Yaskawa INFORM job: SKRZYNIA_4040_-90_STOPNI_10BR.JBI

/JOB
//NAME SKRZYNIA_4040_-90_STOPNI_10BR
///FOLDERNAME 02-SKRZYNIE_JOBS
//POS
///NPOS 404,404,0,30,0,0
///TOOL 0
///POSTYPE PULSE
///PULSE
C00000=0,-52280,40443,0,6876,0
C00001=-82314,-24956,17040,-59626,-27382,-6248
C00002=-93910,-8625,17040,-59626,-43355,-6248
C00003=-98846,-1061,-42166,-80308,-57081,16120
C00004=-100452,6057,-48127,-85711,-56704,21322
C00005=-96957,25597,-37888,-85158,-62082,25522
C00006=-95580,33075,-33256,-84644,-64024,26851
C00007=-94380,33739,-32188,-85134,-63496,26721
C00008=-95580,33075,-33256,-84644,-64024,26851
C00009=-94940,31262,-36138,-85248,-63712,27160
C00010=-95580,33075,-33256,-84644,-64024,26851
C00011=-95263,33142,-33256,-84677,-63995,26850
C00012=-95263,33142,-33256,-84677,-63995,26850
C00013=-94261,33702,-32359,-85087,-63552,26740
C00014=-95263,33142,-33256,-84677,-63995,26850
C00015=-94777,31773,-35433,-85135,-63758,27084
C00016=-95263,33142,-33256,-84677,-63995,26850
C00017=-95260,33144,-33256,-84678,-63995,26850
C00018=-95260,33144,-33256,-84678,-63995,26850
C00019=-94282,33689,-32380,-85076,-63563,26742
C00020=-95260,33144,-33256,-84678,-63995,26850
C00021=-94827,31920,-35204,-85086,-63784,27059
C00022=-95260,33144,-33256,-84678,-63995,26850
C00023=-95258,33145,-33257,-84676,-63996,26846
C00024=-95258,33145,-33257,-84676,-63996,26846
C00025=-94286,33686,-32387,-85074,-63568,26738
C00026=-95258,33145,-33257,-84676,-63996,26846
C00027=-94874,32057,-34990,-85039,-63809,27032
C00028=-95258,33145,-33257,-84676,-63996,26846
C00029=-95377,22848,-19980,-77610,-66139,18413
C00030=-95383,22536,-19091,-77284,-66299,17999
C00031=-94454,23123,-18267,-77513,-65785,17889
C00032=-95383,22536,-19091,-77284,-66299,17999
C00033=-94991,21279,-20843,-77511,-66022,18108
C00034=-95383,22536,-19091,-77284,-66299,17999
C00035=-95258,25631,32269,-66559,-75499,2416
C00036=-95258,25631,32269,-66559,-75499,2416
C00037=-94333,26371,33350,-66433,-74983,2224
C00038=-95258,25631,32269,-66559,-75499,2416
C00039=-94886,24142,30119,-66602,-75133,2534
C00040=-95258,25631,32269,-66559,-75499,2416
C00041=-99189,25294,31874,-88720,-76886,6359
C00042=-99241,29593,38161,-92696,-78880,6430
C00043=-98514,30143,38992,-92642,-78372,6377
C00044=-99241,29593,38161,-92696,-78880,6430
C00045=-98973,29806,38536,-92693,-79698,6341
C00046=-99241,29593,38161,-92696,-78880,6430
C00047=-97871,32974,47728,-100928,-77160,11375
C00048=-97482,34142,50625,-102456,-76680,12291
C00049=-96768,34808,51684,-102358,-76154,12246
C00050=-97504,36083,53738,-102448,-77517,11844
C00051=-97263,35860,53475,-102452,-77986,11780
C00052=-97504,36083,53738,-102448,-77517,11844
C00053=-100410,-1172,-854,-105537,-63273,18802
C00054=-79271,-37169,-30482,-103288,-47510,17696
C00055=-79271,-9415,41877,-76443,-46100,-604
C00056=-100699,17246,57649,-91568,-58011,5122
C00057=-100093,19087,27862,-95634,-72730,8691
C00058=-99472,28508,32136,-95947,-79676,10682
C00059=-98577,29153,33099,-95929,-79046,10644
C00060=-99472,28508,32136,-95947,-79676,10682
C00061=-99113,26771,29576,-96019,-79505,10911
C00062=-99472,28508,32136,-95947,-79676,10682
C00063=-99199,18818,35660,-68259,-73735,6208
C00064=-95720,15423,18785,-70454,-68603,10022
C00065=-95720,15423,18785,-70454,-68603,10022
C00066=-97322,30100,38585,-71742,-79662,10416
C00067=-96349,30901,39804,-71630,-79090,10224
C00068=-97322,30100,38585,-71742,-79662,10416
C00069=-97054,28837,36680,-71776,-79387,10556
C00070=-97322,30100,38585,-71742,-79662,10416
C00071=-97373,30352,38967,-71736,-79717,10385
C00072=-97373,30352,38967,-71736,-79717,10385
C00073=-96432,31128,40151,-71627,-79165,10198
C00074=-97373,30352,38967,-71736,-79717,10385
C00075=-97071,28917,36802,-71776,-79407,10544
C00076=-97373,30352,38967,-71736,-79717,10385
C00077=-97356,30262,38827,-71739,-79698,10398
C00078=-97356,30262,38827,-71739,-79698,10398
C00079=-96507,30957,39891,-71642,-79201,10230
C00080=-97356,30262,38827,-71739,-79698,10398
C00081=-97092,29010,36937,-71773,-79425,10538
C00082=-97356,30262,38827,-71739,-79698,10398
C00083=-99745,23507,8579,-87147,-79275,20063
C00084=-99745,23568,9251,-87081,-79277,19867
C00085=-98882,24102,10002,-87178,-78701,19809
C00086=-99745,23568,9251,-87081,-79277,19867
C00087=-99406,22118,7226,-87176,-79050,20009
C00088=-99745,23568,9251,-87081,-79277,19867
C00089=-99071,22682,8038,-99994,-80807,17980
C00090=-99209,25375,15159,-99348,-81562,16520
C00091=-98424,25891,15901,-99427,-81018,16519
C00092=-99209,25375,15159,-99348,-81562,16520
C00093=-98879,23940,13118,-99425,-81414,16690
C00094=-99209,25375,15159,-99348,-81562,16520
C00095=-97630,34865,50283,-105962,-77348,9129
C00096=-97167,37263,56205,-105494,-76312,8157
C00097=-96392,38071,57532,-105366,-75722,8098
C00098=-97167,37263,56205,-105494,-76312,8157
C00099=-96830,35301,53019,-105613,-76328,8514
C00100=-97167,37263,56205,-105494,-76312,8157
C00101=-98819,19954,1043,-111479,-83154,14713
C00102=-100194,5325,-45038,-118611,-84970,27548
C00103=-77958,-36127,-88985,-138175,-66584,26591
C00104=-62749,-65297,-81682,-146767,-31843,20298
C00105=-53629,-59560,-53714,-89083,-24254,-4356
C00106=-73187,-23116,26488,-26118,-57509,-28469
C00107=-96139,-22548,-25766,-67560,-51232,-5154
C00108=-98398,-8109,-25057,-81551,-55130,4513
C00109=-99451,17861,2757,-80571,-73406,6045
C00110=-99056,24650,11359,-80216,-77425,5946
C00111=-98115,25261,12228,-80295,-76818,5843
C00112=-99056,24650,11359,-80216,-77425,5946
C00113=-98800,23560,9817,-80291,-77224,6050
C00114=-99056,24650,11359,-80216,-77425,5946
C00115=-99819,33446,48735,-87787,-79679,-1235
C00116=-99819,33446,48735,-87787,-79679,-1235
C00117=-98945,34179,49898,-87659,-79086,-1350
C00118=-99819,33446,48735,-87787,-79679,-1235
C00119=-99591,32133,46677,-87830,-79529,-1033
C00120=-99819,33446,48735,-87787,-79679,-1235
C00121=-98841,-14263,-23955,-101504,-55644,8170
C00122=-96175,-21848,-39130,-108881,-63715,10829
C00123=-56537,-51855,-41447,-79827,-26849,-3300
///LIMIT ON
C00124=-37962,-64638,6899,-31784,1461,6885
///LIMIT OFF
C00125=0,-43112,23163,32261,-40956,29092
C00126=-38075,-37396,2384,-17964,-21120,46852
C00127=-50509,-19000,10610,-51503,-15997,61182
C00128=-53130,-17211,12007,-56251,-17152,63186
C00129=-51822,-15992,12994,-55136,-16324,62798
C00130=-53635,-15431,13457,-57815,-17251,63894
C00131=-53130,-17211,12007,-56251,-17152,63186
C00132=-50704,-18403,11069,-52157,-16018,61478
C00133=-53231,-16470,14622,-53206,-17893,61673
C00134=-51756,-15101,15744,-51790,-16990,61165
C00135=-53741,-14453,16285,-54808,-17949,62397
C00136=-53231,-17580,11714,-56182,-17246,63139
C00137=-51814,-19410,10295,-53186,-16720,61844
C00138=-53629,-18979,7405,-62018,-16535,65958
C00139=-52238,-17698,8415,-61175,-15613,65699
C00140=-53551,-17401,8655,-62910,-16346,66402
C00141=-52880,-17654,11656,-55678,-17066,62935
C00142=-51005,-17995,11387,-52847,-16122,61778
C00143=-52964,-17611,11689,-55811,-17106,62990
C00144=-51611,-16353,12697,-54642,-16249,62582
C00145=-53495,-15765,13180,-57466,-17201,63739
C00146=-52964,-17611,11689,-55811,-17106,62990
C00147=-51030,-17982,11395,-52891,-16135,61798
C00148=-52975,-17563,11726,-55850,-17109,63009
C00149=-51607,-16289,12749,-54669,-16241,62596
C00150=-53283,-15811,13140,-57177,-17094,63622
C00151=-52975,-17563,11726,-55850,-17109,63009
C00152=-50945,-18019,11363,-52741,-16103,61737
C00153=-52728,-17788,11545,-55393,-17010,62816
C00154=-51045,-16207,12813,-53894,-15944,62287
C00155=-52895,-15647,13274,-56746,-16874,63461
C00156=-52728,-17788,11545,-55393,-17010,62816
C00157=-50945,-18019,11363,-52741,-16103,61737
C00158=-52556,-17520,11756,-55311,-16888,62798
C00159=-51113,-16157,12849,-54025,-15975,62343
C00160=-52730,-15718,13210,-56498,-16792,63358
C00161=-52556,-17520,11756,-55311,-16888,62798
C00162=-50945,-18019,11363,-52741,-16103,61737
C00163=-51893,-17787,11546,-54246,-16568,62356
C00164=-50379,-16341,12703,-52826,-15610,61849
C00165=-52406,-15704,13225,-56071,-16614,63190
C00166=-51893,-17787,11546,-54246,-16568,62356
C00167=-50028,-22953,-3957,-22347,-31919,54220
C00168=-50947,-22502,-3625,-23433,-32061,54736
C00169=-49421,-20951,-2455,-21951,-31329,54057
C00170=-51207,-20433,-2055,-24026,-31698,55041
C00171=-50529,-22709,-3778,-22940,-31995,54502
C00172=-49763,-25421,-36239,-24565,-26935,60445
C00173=-49763,-25421,-36239,-24565,-26935,60445
C00174=-48299,-23485,-34758,-23276,-26122,59713
C00175=-50218,-22723,-34165,-25568,-26529,60993
C00176=-49763,-25421,-36239,-24565,-26935,60445
C00177=-50713,-12366,-58367,-41124,-17813,74400
C00178=-50824,-12254,-58263,-41255,-17847,74484
C00179=-49431,-10052,-56192,-40383,-17131,73813
C00180=-50915,-9358,-55524,-41955,-17664,74847
C00181=-51028,-12852,-58814,-41301,-17980,74542
C00182=-49763,-25421,-36239,-24565,-26935,60445
C00183=-50529,-22709,-3778,-22940,-31995,54502
C00184=-45389,-28224,4312,-35967,-15579,54278
C00185=-40154,-51179,-915,-24203,-8234,36524
C00186=0,-52280,40443,0,6876,0
C00187=-41463,-32191,18163,-91991,-64949,55938
C00188=0,-52277,40442,0,6872,4
C00189=-82314,-24956,17040,-59626,-27382,-6248
C00190=-93910,-8625,17040,-59626,-43355,-6248
C00191=-98846,-1061,-42166,-80308,-57081,16120
C00192=-100452,6057,-48127,-85711,-56704,21322
C00193=-95564,34698,-34234,-85516,-63941,27819
C00194=-94221,34299,-28769,-82558,-65564,25844
C00195=-94107,37241,-30442,-84005,-65307,27544
C00196=-95103,32620,-31323,-83378,-64939,26072
C00197=-95103,32620,-31323,-83378,-64939,26072
C00198=-93990,32828,-31380,-83932,-64473,26160
C00199=-94063,31710,-30585,-83283,-64598,25457
C00200=-96692,32939,-31211,-82617,-65723,26190
C00201=-96111,21840,170,-71736,-70232,11396
C00202=-94229,22391,773,-71789,-70557,11468
C00203=-94283,22521,1025,-71678,-70686,11433
C00204=-95675,19167,-4176,-72970,-68231,11735
C00205=-95681,24338,3488,-71459,-71669,11415
C00206=-94245,22750,1246,-71757,-70674,11453
C00207=-94341,22923,1499,-71729,-70746,11440
C00208=-96213,24222,3324,-71394,-71999,11479
C00209=-95517,23330,2066,-71543,-71508,11507
C00210=-94304,22892,1449,-71738,-70721,11443
C00211=-94158,22889,1452,-71756,-70627,11429
C00212=-96071,24319,3461,-71408,-71916,11455
C00213=-96941,-6406,-33809,-76117,-54125,10511
C00214=-90643,-26862,-25633,-62597,-56791,-1368
C00215=-66103,-61757,7450,-21008,-32955,-5749
C00216=4223,-52290,40457,-5766,6913,3980
C00217=4223,-52290,40457,-5766,6913,3980
C00218=-4825,-36686,24602,37792,-30278,35378
C00219=-46221,-29633,7403,-27051,-24124,46751
C00220=-46221,-29633,7403,-27051,-24124,46751
C00221=-52474,-20611,11454,-41004,-23045,52959
C00222=-60257,-19980,-2088,-84190,-23320,82051
C00223=-63868,-19883,-6318,-95759,-28031,88346
C00224=-51819,-22965,8574,-41365,-22900,53139
C00225=-4825,-36686,24602,37792,-30278,35378
C00226=0,-52280,40443,0,6876,0
C00227=4223,-52290,40457,-5766,6913,3980
C00228=-66103,-61757,7450,-21008,-32955,-5749
C00229=-89093,-33107,-44597,-67545,-52550,2722
C00230=-96941,-6406,-33809,-76117,-54125,10511
C00231=-99429,14378,84,-80785,-71596,8628
C00232=-99699,24313,24829,-82602,-77917,4569
C00233=-98066,26841,20697,-83331,-79245,6860
C00234=-98079,26929,20513,-83349,-79351,6953
C00235=-99638,19663,10292,-84193,-74452,7551
C00236=-98909,20891,5205,-92499,-77779,3679
C00237=-97991,21897,3469,-96150,-79490,1870
C00238=-97094,22407,2872,-101449,-80737,3094
C00239=-98052,22735,7381,-100906,-80646,1724
C00240=-96016,28471,32512,-109475,-77029,-270
C00241=-93697,27731,31018,-109675,-75757,229
C00242=-93697,30712,42128,-108463,-73689,-2160
C00243=-100174,9543,-9646,-113455,-77250,7387
C00244=-100174,1289,-12558,-103866,-68626,6781
C00245=-100177,-4656,-30138,-114506,-71921,12431
C00246=-97546,-19067,-24950,-97028,-60115,5718
C00247=-61441,-38616,11032,-55510,-42874,-3049
C00248=4223,-52290,40457,-5766,6913,3980
C00249=4223,-52290,40457,-5766,6913,3980
C00250=-4825,-36686,24602,37792,-30278,35378
C00251=-46221,-29633,7403,-27051,-24124,46751
C00252=-56796,-22932,368,-68953,-21567,70907
C00253=-61611,-20349,-6598,-95791,-25091,88405
C00254=-62244,-19942,-5791,-95984,-25882,88372
C00255=-57752,-2938,32150,-100764,-20307,82364
C00256=-58257,-11045,22458,-94361,-23082,79795
C00257=-49294,-34086,9663,-30689,-30758,52546
C00258=4223,-52290,40457,-5766,6913,3980
C00259=0,-52280,40443,0,6876,0
C00260=0,-52280,40443,0,6876,0
C00261=-61754,-61602,7279,-16215,-32140,-7126
C00262=-89313,-24027,20291,-53466,-58905,-4975
C00263=-97807,-25409,-21837,-78881,-62828,2121
C00264=-100103,-15040,-13507,-79140,-58253,2724
C00265=-99725,9645,23361,-67154,-68568,-2059
C00266=-99271,16305,34765,-72797,-70067,-2351
C00267=-98402,25140,29245,-92090,-76944,4625
C00268=-98402,28265,40696,-90956,-76523,2010
C00269=-98754,23130,28932,-98122,-73671,5428
C00270=-98112,-9349,-13739,-99107,-55531,8873
C00271=-87692,-34175,-39658,-96739,-43399,8225
C00272=-75165,-16680,32803,-38944,-52307,-27215
C00273=-75165,-16680,32803,-38944,-52307,-27215
C00274=-96391,11374,61850,-52875,-60261,-22353
C00275=-96391,-17993,-25254,-79577,-45337,-1997
C00276=-84714,-13514,-21320,-79690,-37366,-2300
C00277=-92093,-5454,-13554,-80916,-52292,-613
C00278=-99761,24721,23429,-79408,-77929,-316
C00279=-99564,24916,23930,-79374,-77823,-417
C00280=-100005,27069,23687,-81767,-79755,895
C00281=-97295,30454,38512,-73622,-79542,-3831
C00282=-98471,27958,25022,-81751,-79627,782
C00283=-99805,23386,18402,-82055,-77455,1200
C00284=-100093,24719,20298,-81968,-77939,1081
C00285=-98451,26404,20171,-83400,-79044,-389
C00286=-98528,26732,19657,-84000,-79459,-654
C00287=-100109,23919,19160,-82044,-77303,1139
C00288=-98037,-4340,-16930,-86109,-58746,2389
C00289=-93345,-31758,-40240,-83703,-37467,-946
C00290=-81087,-35886,-14825,-53529,-36311,-18004
C00291=-47029,-49867,-20464,-11808,-29290,-36568
///LIMIT ON
C00292=-41431,-67449,10869,-1325,127,-6150
///LIMIT OFF
C00293=6328,-52297,40483,-8599,6957,5944
C00294=6328,-52297,40483,-8599,6957,5944
C00295=-10231,-60460,6271,71658,-11927,-13637
C00296=-49129,-39322,3023,-34904,-18609,43900
C00297=-57258,-19535,13114,-46502,-25798,55150
C00298=-58736,-19151,1344,-78268,-22199,76919
C00299=-56868,-17231,8572,-62431,-21728,66645
C00300=-56011,-29317,6725,-41009,-27363,52457
C00301=-10137,-60963,4526,62308,-14518,-6745
C00302=0,-52280,40443,0,6876,0
C00303=0,-52280,40443,0,6876,0
C00304=-41653,-63035,2931,-3578,-7576,-14589
C00305=-45770,-50109,-20524,-10089,-29273,-37310
C00306=-80544,-36303,-15042,-52975,-36116,-18265
C00307=-93028,-32302,-40599,-83495,-37263,-1079
C00308=-98446,-3141,-15678,-86094,-59021,2414
C00309=-99951,24070,19376,-82000,-77829,1145
C00310=-98655,27908,24922,-81730,-79774,792
C00311=-98593,28720,26118,-81685,-80145,709
C00312=-99951,24070,19376,-82000,-77829,1145
C00313=-99951,24070,19376,-82000,-77829,1145
C00314=-98577,27118,23759,-81796,-79157,859
C00315=-98518,28577,26461,-81649,-79882,537
C00316=-99951,24070,19376,-82000,-77829,1145
C00317=-100023,27130,33022,-92975,-78123,-161
C00318=-98580,26185,31637,-93003,-77167,-1
C00319=-98580,30404,46303,-91600,-76541,-3267
C00320=-100724,18056,24349,-92081,-73134,-455
C00321=-98404,-4962,-6255,-93190,-58383,1895
C00322=-99487,-12045,-28221,-93829,-57357,5545
C00323=-95086,-30272,-46998,-91958,-53375,4609
C00324=-81694,-37220,-20464,-64791,-45723,-12569
C00325=-45770,-50109,-20524,-10089,-29273,-37310
///LIMIT ON
C00326=-40984,-65135,6743,-2520,-4051,-10897
///LIMIT OFF
C00327=0,-52280,40443,0,6876,0
C00328=0,-52280,40443,0,6876,0
///LIMIT ON
C00329=-50974,-46557,23391,-77768,-13896,42026
///LIMIT OFF
C00330=-53474,-39983,4253,-39182,-18848,44272
C00331=-56619,-19856,12878,-45665,-25558,54806
C00332=-53298,-26712,-11188,-26889,-32979,52528
C00333=-57200,-20845,-7559,-37425,-33513,53351
C00334=-58648,-23818,-25853,-45100,-31207,62168
C00335=-58477,-22145,-38977,-48305,-29254,64725
C00336=-51868,-27423,-11673,-25269,-32728,51737
C00337=-49121,-45409,-2608,-26656,-19965,38583
C00338=-21301,-61008,4568,43957,-10534,-712
C00339=0,-52280,40443,0,6876,0
C00340=0,-52280,40443,0,6876,0
///LIMIT ON
C00341=-40221,-67507,11044,-1325,-65,-6716
///LIMIT OFF
C00342=-45770,-50109,-20525,-10088,-29274,-37311
C00343=-80544,-36303,-15042,-52975,-36116,-18265
C00344=-93028,-32301,-40599,-83495,-37262,-1079
C00345=-97841,-4898,-17503,-86112,-58614,2374
C00346=-97574,22325,42435,-102650,-66613,-1893
C00347=-95754,35899,57018,-103970,-74003,-2798
C00348=-95754,43745,77672,-101743,-71699,-6650
C00349=-99714,17597,9613,-108150,-76803,6279
C00350=-93796,-17226,-33718,-118170,-55432,13587
C00351=-66816,-54797,-57006,-119089,-33370,13303
C00352=-66816,-52758,-50486,-115256,-31854,11154
C00353=-98141,-7636,2315,-105626,-50514,3722
C00354=-99521,20918,46679,-89083,-66665,-5358
C00355=-98691,34973,58126,-90608,-76643,-4580
C00356=-98691,42061,76615,-89053,-76304,-8086
C00357=-98720,15018,65588,-59406,-66947,-17238
C00358=-93628,-24224,-10838,-81898,-52333,-4131
C00359=-86170,-37737,-28198,-69261,-47898,-9342
C00360=-45770,-50109,-20525,-10088,-29274,-37311
///LIMIT ON
C00361=-40221,-67507,11044,-1325,-65,-6716
///LIMIT OFF
C00362=0,-52280,40443,0,6876,0
C00363=0,-52280,40443,0,6876,0
///LIMIT ON
C00364=-50971,-46557,23390,-77766,-13895,42026
///LIMIT OFF
C00365=-53475,-39984,4253,-39182,-18848,44273
C00366=-56619,-19856,12878,-45665,-25558,54806
C00367=-57643,-27958,-8553,-51854,-24771,59787
C00368=-66195,-24410,-19095,-90567,-31132,85904
C00369=-63290,-24193,-14362,-80030,-27547,78073
C00370=-39040,-40975,-15408,-18643,-21575,44866
C00371=-11647,-69843,-10959,56399,-11165,-4616
C00372=-15394,-57237,30542,-10392,5525,8219
C00373=0,-52280,40443,0,6876,0
C00374=0,-52280,40443,0,6876,0
///LIMIT ON
C00375=-40221,-67507,11044,-1325,-65,-6716
///LIMIT OFF
C00376=-45770,-50109,-20525,-10088,-29274,-37311
C00377=-95022,-19559,-3970,-66108,-42168,-11789
C00378=-84972,-7110,7117,-67721,-41324,-10731
C00379=-83869,-8155,6098,-67213,-40658,-10968
C00380=-99927,23961,20220,-85683,-78298,772
C00381=-98562,26853,28284,-85090,-78334,-823
C00382=-98562,24944,18750,-86001,-78172,1594
C00383=-99530,24174,17652,-85964,-78826,1685
C00384=-98491,25445,31196,-89357,-76395,-673
C00385=-98197,26014,32882,-93044,-76072,-339
C00386=-99839,23064,19027,-85806,-76881,822
C00387=-86774,-13232,-16630,-85484,-41019,-1154
C00388=-97999,-21060,-29835,-88214,-48653,956
C00389=-98846,-3268,25064,-74217,-51189,-12584
C00390=-70313,-35289,-4922,-51188,-38634,-20596
C00391=-81694,-37221,-20464,-64791,-45723,-12569
C00392=-45770,-50109,-20525,-10088,-29274,-37311
C00393=-41628,-63095,3038,-3547,-7472,-14475
C00394=4223,-52290,40457,-5766,6913,3980
///LIMIT ON
C00395=-50971,-46557,23390,-77766,-13895,42026
///LIMIT OFF
C00396=-53475,-39984,4253,-39182,-18848,44273
C00397=-56619,-19856,12878,-45665,-25558,54806
C00398=-53891,-17708,14512,-43170,-23995,53902
C00399=-60674,-17500,6427,-71116,-24772,71097
C00400=-63181,-17997,2063,-82122,-26831,78394
C00401=-39402,-27697,7664,-17904,-21663,43170
C00402=-11647,-69843,-10959,56399,-11165,-4616
C00403=0,-52280,40443,0,6876,0
BC00000=372198
BC00001=352964
BC00002=352964
BC00003=406723
BC00004=352964
BC00005=352964
BC00006=352964
BC00007=352964
BC00008=352964
BC00009=352964
BC00010=352964
BC00011=399066
BC00012=399066
BC00013=399066
BC00014=399066
BC00015=399066
BC00016=399066
BC00017=445276
BC00018=445276
BC00019=445276
BC00020=445276
BC00021=445276
BC00022=445276
BC00023=491380
BC00024=491380
BC00025=491380
BC00026=491380
BC00027=491380
BC00028=491380
BC00029=481377
BC00030=480887
BC00031=480887
BC00032=480887
BC00033=480888
BC00034=480887
BC00035=467227
BC00036=467227
BC00037=467227
BC00038=467227
BC00039=467227
BC00040=467227
BC00041=464142
BC00042=463563
BC00043=463563
BC00044=463563
BC00045=463563
BC00046=463563
BC00047=467130
BC00048=467852
BC00049=467852
BC00050=467852
BC00051=467852
BC00052=467852
BC00053=431056
BC00054=431056
BC00055=478309
BC00056=512702
BC00057=523223
BC00058=534753
BC00059=534753
BC00060=534753
BC00061=534753
BC00062=534753
BC00063=621951
BC00064=621951
BC00065=621951
BC00066=621951
BC00067=621951
BC00068=621951
BC00069=621951
BC00070=621951
BC00071=645037
BC00072=645037
BC00073=645037
BC00074=645037
BC00075=645037
BC00076=645037
BC00077=691109
BC00078=691109
BC00079=691109
BC00080=691109
BC00081=691109
BC00082=691109
BC00083=714198
BC00084=714198
BC00085=714197
BC00086=714198
BC00087=714198
BC00088=714198
BC00089=721422
BC00090=721422
BC00091=721422
BC00092=721422
BC00093=721422
BC00094=721422
BC00095=705839
BC00096=705839
BC00097=705839
BC00098=705839
BC00099=705839
BC00100=705839
BC00101=706227
BC00102=715152
BC00103=741215
BC00104=815410
BC00105=809921
BC00106=799182
BC00107=831839
BC00108=838454
BC00109=838479
BC00110=838485
BC00111=838485
BC00112=838485
BC00113=838485
BC00114=838485
BC00115=819448
BC00116=834809
BC00117=834809
BC00118=834809
BC00119=834809
BC00120=834809
BC00121=835662
BC00122=825379
BC00123=817159
BC00124=681039
BC00125=719629
BC00126=804722
BC00127=797458
BC00128=797458
BC00129=797458
BC00130=797458
BC00131=797458
BC00132=736016
BC00133=736016
BC00134=736016
BC00135=736016
BC00136=736016
BC00137=674586
BC00138=674586
BC00139=674586
BC00140=674586
BC00141=674586
BC00142=613184
BC00143=613184
BC00144=613184
BC00145=613184
BC00146=613184
BC00147=551699
BC00148=551699
BC00149=551699
BC00150=551699
BC00151=551699
BC00152=490298
BC00153=490298
BC00154=490298
BC00155=490298
BC00156=490298
BC00157=428826
BC00158=428826
BC00159=428826
BC00160=428826
BC00161=428826
BC00162=367374
BC00163=367374
BC00164=367374
BC00165=367374
BC00166=367374
BC00167=367378
BC00168=367378
BC00169=367378
BC00170=367378
BC00171=367378
BC00172=367378
BC00173=367378
BC00174=367378
BC00175=367378
BC00176=367378
BC00177=367378
BC00178=367378
BC00179=367378
BC00180=367378
BC00181=367378
BC00182=367378
BC00183=367378
BC00184=367374
BC00185=441050
BC00186=441050
BC00187=791478
BC00188=382983
BC00189=352964
BC00190=352964
BC00191=408260
BC00192=352964
BC00193=352964
BC00194=353544
BC00195=352960
BC00196=353556
BC00197=391964
BC00198=400011
BC00199=389600
BC00200=400107
BC00201=381081
BC00202=388397
BC00203=381081
BC00204=388818
BC00205=427172
BC00206=434877
BC00207=427169
BC00208=427169
BC00209=457913
BC00210=457913
BC00211=450237
BC00212=450041
BC00213=414344
BC00214=450041
BC00215=427058
BC00216=450041
BC00217=400994
BC00218=490644
BC00219=563016
BC00220=563016
BC00221=563016
BC00222=563016
BC00223=624162
BC00224=624476
BC00225=490644
BC00226=400994
BC00227=450041
BC00228=450041
BC00229=413692
BC00230=498778
BC00231=464973
BC00232=451598
BC00233=459057
BC00234=451696
BC00235=459288
BC00236=477534
BC00237=485795
BC00238=485795
BC00239=485795
BC00240=461742
BC00241=461742
BC00242=461742
BC00243=461742
BC00244=464778
BC00245=461044
BC00246=455085
BC00247=441558
BC00248=492251
BC00249=528027
BC00250=720637
BC00251=795617
BC00252=805108
BC00253=808590
BC00254=827541
BC00255=790719
BC00256=786930
BC00257=760893
BC00258=450041
BC00259=450041
BC00260=450041
BC00261=450041
BC00262=509147
BC00263=545841
BC00264=541316
BC00265=532881
BC00266=530910
BC00267=529272
BC00268=529272
BC00269=529176
BC00270=533263
BC00271=538121
BC00272=540993
BC00273=589567
BC00274=589567
BC00275=648537
BC00276=648537
BC00277=648537
BC00278=648537
BC00279=617841
BC00280=617841
BC00281=611605
BC00282=617971
BC00283=617841
BC00284=634993
BC00285=633229
BC00286=640873
BC00287=640937
BC00288=640937
BC00289=640937
BC00290=640937
BC00291=640937
BC00292=640937
BC00293=640937
BC00294=528027
BC00295=469376
BC00296=406602
BC00297=315730
BC00298=315726
BC00299=376881
BC00300=377231
BC00301=431999
BC00302=431999
BC00303=640937
BC00304=640937
BC00305=640937
BC00306=640937
BC00307=640937
BC00308=640937
BC00309=679258
BC00310=679258
BC00311=687013
BC00312=679258
BC00313=702338
BC00314=702338
BC00315=709052
BC00316=702338
BC00317=697065
BC00318=697065
BC00319=697065
BC00320=699422
BC00321=702188
BC00322=721854
BC00323=728490
BC00324=748432
BC00325=703131
BC00326=649416
BC00327=640936
BC00328=580559
BC00329=483911
BC00330=372992
BC00331=315730
BC00332=315730
BC00333=315730
BC00334=315730
BC00335=315730
BC00336=315730
BC00337=379280
BC00338=431999
BC00339=431999
BC00340=640937
BC00341=640937
BC00342=640937
BC00343=640937
BC00344=640937
BC00345=640937
BC00346=690236
BC00347=698481
BC00348=698481
BC00349=700031
BC00350=700031
BC00351=700031
BC00352=758299
BC00353=758299
BC00354=755546
BC00355=768208
BC00356=768208
BC00357=768208
BC00358=750310
BC00359=761341
BC00360=703131
BC00361=640937
BC00362=640937
BC00363=580559
BC00364=483911
BC00365=421515
BC00366=442691
BC00367=465804
BC00368=465286
BC00369=526143
BC00370=526236
BC00371=526236
BC00372=526236
BC00373=526236
BC00374=640937
BC00375=640937
BC00376=823629
BC00377=816144
BC00378=816144
BC00379=816144
BC00380=839508
BC00381=839510
BC00382=839510
BC00383=839510
BC00384=839617
BC00385=839617
BC00386=840477
BC00387=836719
BC00388=828295
BC00389=807430
BC00390=790908
BC00391=748432
BC00392=703131
BC00393=656709
BC00394=640937
BC00395=657676
BC00396=664515
BC00397=684473
BC00398=684473
BC00399=684473
BC00400=746207
BC00401=745829
BC00402=704594
BC00403=650116
///POSTYPE BASE
///RECTAN
///RCONF 1,0,0,0,0,0,0,0,0,0,0,0,0,0,0,0,0,0,0,0,0,0,0,0
P00006=0.000,0.000,0.000,0.0000,0.0000,0.0000
///RCONF 0,0,0,0,0,0,0,0,0,0,0,0,0,0,0,0,0,0,0,0,0,0,0,0
P00058=0.000,0.000,3.000,0.0000,0.0000,0.0000
///RCONF 1,0,0,0,0,0,0,0,0,0,0,0,0,0,0,0,0,0,0,0,0,0,0,0
P00300=-0.036,-1.505,2.318,0.0000,0.0000,0.0000
P00301=0.046,-2.112,7.779,0.0000,0.0000,0.0000
P00302=-0.180,-2.409,6.326,0.0000,0.0000,0.0000
///RCONF 0,0,0,0,0,0,0,0,0,0,0,0,0,0,0,0,0,0,0,0,0,0,0,0
P00303=-0.004,-1.437,-4.584,0.0000,0.0000,0.0000
P00304=0.028,-1.666,-4.234,0.0000,0.0000,0.0000
P00305=-0.003,-1.920,-3.501,0.0000,0.0000,0.0000
P00306=0.015,-2.252,-3.054,0.0000,0.0000,0.0000
P00307=0.019,-2.151,-5.077,0.0000,0.0000,0.0000
P00308=-0.003,-2.092,-4.888,0.0000,0.0000,0.0000
P00309=-0.040,-2.205,-4.992,0.0000,0.0000,0.0000
P00310=-0.006,-2.490,-5.925,0.0000,0.0000,0.0000
P00311=-0.007,-2.079,-5.307,0.0000,0.0000,0.0000
P00312=-0.032,2.202,-7.632,0.0000,0.0000,0.0000
///RCONF 1,0,0,0,0,0,0,0,0,0,0,0,0,0,0,0,0,0,0,0,0,0,0,0
P00313=-0.088,1.055,2.110,0.0000,0.0000,0.0000
P00314=-0.055,1.752,1.634,0.0000,0.0000,0.0000
P00316=0.009,2.112,2.075,0.0000,0.0000,0.0000
P00317=-0.015,2.781,3.126,0.0000,0.0000,0.0000
///RCONF 0,0,0,0,0,0,0,0,0,0,0,0,0,0,0,0,0,0,0,0,0,0,0,0
P00351=13.563,-0.027,-0.653,0.0000,0.0000,0.0000
P00352=13.252,-0.027,-0.827,0.0000,0.0000,0.0000
P00353=10.971,-0.082,0.776,0.0000,0.0000,0.0000
P00354=-0.024,2.508,-1.824,0.0000,0.0000,0.0000
P00355=-0.001,2.528,-1.131,0.0000,0.0000,0.0000
P00356=-0.034,2.921,-0.262,0.0000,0.0000,0.0000
P00357=0.003,3.386,-0.091,0.0000,0.0000,0.0000
P00358=0.014,3.037,-0.020,0.0000,0.0000,0.0000
P00359=-0.005,2.731,0.912,0.0000,0.0000,0.0000
P00360=-0.011,3.412,0.438,0.0000,0.0000,0.0000
P00361=0.018,3.050,1.253,0.0000,0.0000,0.0000
//INST
///DATE 2025/03/25 11:13
///ATTR SC,RW
///GROUP1 RB1,BS1
NOP
CALL JOB:MOVE_INTO_TUNNEL
MOVJ C00000 BC00000 VJ=50.00
MOVJ C00001 BC00001 VJ=40.00
MOVJ C00002 BC00002 VJ=40.00
MOVL C00003 BC00003 V=666.7
COMM MOVJ C00004 BC00004 VJ=30.00
COMM MOVL C00005 BC00005 V=500.0
COMM '------------------------
COMM 'W31.2
COMM '------------------------
COMM MOVL C00006 BC00006 V=166.7 PL=0
COMM REFP 3 C00007 BC00007
COMM CALL JOB:SEARCH-R1
COMM SET P0300 P0006
COMM SFTON P0300
COMM MOVL C00008 BC00008 V=166.7 PL=0
COMM REFP 3 C00009 BC00009
COMM CALL JOB:SEARCH-R1
COMM SET P0300 P0006
COMM SFTON P0300
COMM MOVL C00010 BC00010 V=166.7 PL=0
COMM SFTOF
COMM '------------------------
COMM 'W31.4
COMM '------------------------
COMM MOVL C00011 BC00011 V=500.0
COMM MOVL C00012 BC00012 V=166.7 PL=0
COMM REFP 3 C00013 BC00013
COMM CALL JOB:SEARCH-R1
COMM SET P0301 P0006
COMM SFTON P0301
COMM MOVL C00014 BC00014 V=166.7 PL=0
COMM REFP 3 C00015 BC00015
COMM CALL JOB:SEARCH-R1
COMM SET P0301 P0006
COMM SFTON P0301
COMM MOVL C00016 BC00016 V=166.7 PL=0
COMM SFTOF
'------------------------
'W31.6
'------------------------
MOVL C00017 BC00017 V=500.0
MOVL C00018 BC00018 V=166.7 PL=0
REFP 3 C00019 BC00019
CALL JOB:SEARCH-R1
SET P0302 P0006
SFTON P0302
MOVL C00020 BC00020 V=166.7 PL=0
REFP 3 C00021 BC00021
CALL JOB:SEARCH-R1
SET P0302 P0006
SFTON P0302
MOVL C00022 BC00022 V=166.7 PL=0
SFTOF
'------------------------
'W31.8
'------------------------
MOVL C00023 BC00023 V=500.0
MOVL C00024 BC00024 V=166.7 PL=0
REFP 3 C00025 BC00025
CALL JOB:SEARCH-R1
SET P0303 P0006
SFTON P0303
MOVL C00026 BC00026 V=166.7 PL=0
REFP 3 C00027 BC00027
CALL JOB:SEARCH-R1
SET P0303 P0006
SFTON P0303
MOVL C00028 BC00028 V=166.7 PL=0
SFTOF
'------------------------
'W31.9
'------------------------
MOVL C00029 BC00029 V=500.0
MOVL C00030 BC00030 V=166.7 PL=0
REFP 3 C00031 BC00031
CALL JOB:SEARCH-R1
SET P0304 P0006
SFTON P0304
MOVL C00032 BC00032 V=166.7 PL=0
REFP 3 C00033 BC00033
CALL JOB:SEARCH-R1
SET P0304 P0006
SFTON P0304
MOVL C00034 BC00034 V=166.7 PL=0
SFTOF
'------------------------
'W31.11
'------------------------
MOVL C00035 BC00035 V=500.0
MOVL C00036 BC00036 V=166.7 PL=0
REFP 3 C00037 BC00037
CALL JOB:SEARCH-R1
SET P0305 P0006
SFTON P0305
MOVL C00038 BC00038 V=166.7 PL=0
REFP 3 C00039 BC00039
CALL JOB:SEARCH-R1
SET P0305 P0006
SFTON P0305
MOVL C00040 BC00040 V=166.7 PL=0
SFTOF
'------------------------
'W31.13
'------------------------
MOVL C00041 BC00041 V=500.0
MOVL C00042 BC00042 V=166.7 PL=0
REFP 3 C00043 BC00043
CALL JOB:SEARCH-R1
SET P0306 P0006
SFTON P0306
MOVL C00044 BC00044 V=166.7 PL=0
REFP 3 C00045 BC00045
CALL JOB:SEARCH-R1
SET P0306 P0006
SFTON P0306
MOVL C00046 BC00046 V=166.7 PL=0
SFTOF
'------------------------
'W31.14
'------------------------
MOVL C00047 BC00047 V=333.3
MOVL C00048 BC00048 V=166.7 PL=0
REFP 3 C00049 BC00049
CALL JOB:SEARCH-R1
SET P0307 P0006
SFTON P0307
MOVL C00050 BC00050 V=166.7 PL=0
REFP 3 C00051 BC00051
CALL JOB:SEARCH-R1
SET P0307 P0006
SFTON P0307
MOVL C00052 BC00052 V=166.7 PL=0
SFTOF
MOVL C00053 BC00053 V=500.0
MOVL C00054 BC00054 V=500.0
MOVL C00055 BC00055 V=500.0
MOVL C00056 BC00056 V=500.0
'------------------------
'W31.16
'------------------------
MOVL C00057 BC00057 V=500.0
MOVL C00058 BC00058 V=166.7 PL=0
REFP 3 C00059 BC00059
CALL JOB:SEARCH-R1
SET P0308 P0006
SFTON P0308
MOVL C00060 BC00060 V=166.7 PL=0
REFP 3 C00061 BC00061
CALL JOB:SEARCH-R1
SET P0308 P0006
SFTON P0308
MOVL C00062 BC00062 V=166.7 PL=0
SFTOF
MOVL C00063 BC00063 V=500.0
MOVL C00064 BC00064 V=333.3
'------------------------
'W31.18
'------------------------
MOVL C00065 BC00065 V=166.7
MOVL C00066 BC00066 V=133.3 PL=0
REFP 3 C00067 BC00067
CALL JOB:SEARCH-R1
SET P0309 P0006
SFTON P0309
MOVL C00068 BC00068 V=66.7 PL=0
REFP 3 C00069 BC00069
CALL JOB:SEARCH-R1
SET P0309 P0006
SFTON P0309
MOVL C00070 BC00070 V=66.7 PL=0
SFTOF
'------------------------
'W31.19
'------------------------
MOVL C00071 BC00071 V=500.0
MOVL C00072 BC00072 V=166.7 PL=0
REFP 3 C00073 BC00073
CALL JOB:SEARCH-R1
SET P0310 P0006
SFTON P0310
MOVL C00074 BC00074 V=166.7 PL=0
REFP 3 C00075 BC00075
CALL JOB:SEARCH-R1
SET P0310 P0006
SFTON P0310
MOVL C00076 BC00076 V=166.7 PL=0
SFTOF
'------------------------
'W31.21
'------------------------
MOVL C00077 BC00077 V=500.0
MOVL C00078 BC00078 V=166.7 PL=0
REFP 3 C00079 BC00079
CALL JOB:SEARCH-R1
SET P0311 P0006
SFTON P0311
MOVL C00080 BC00080 V=166.7 PL=0
REFP 3 C00081 BC00081
CALL JOB:SEARCH-R1
SET P0311 P0006
SFTON P0311
MOVL C00082 BC00082 V=166.7 PL=0
SFTOF
'------------------------
'W31.22
'------------------------
MOVL C00083 BC00083 V=500.0
MOVL C00084 BC00084 V=166.7 PL=0
REFP 3 C00085 BC00085
CALL JOB:SEARCH-R1
SET P0312 P0006
SFTON P0312
MOVL C00086 BC00086 V=166.7 PL=0
REFP 3 C00087 BC00087
CALL JOB:SEARCH-R1
SET P0312 P0006
SFTON P0312
MOVL C00088 BC00088 V=166.7 PL=0
SFTOF
'------------------------
'W31.24
'------------------------
MOVL C00089 BC00089 V=500.0
MOVL C00090 BC00090 V=166.7 PL=0
REFP 3 C00091 BC00091
CALL JOB:SEARCH-R1
SET P0313 P0006
SFTON P0313
MOVL C00092 BC00092 V=166.7 PL=0
REFP 3 C00093 BC00093
CALL JOB:SEARCH-R1
SET P0313 P0006
SFTON P0313
MOVL C00094 BC00094 V=166.7 PL=0
SFTOF
'------------------------
'W31.26
'------------------------
MOVL C00095 BC00095 V=500.0
MOVL C00096 BC00096 V=166.7 PL=0
REFP 3 C00097 BC00097
CALL JOB:SEARCH-R1
SET P0314 P0006
SFTON P0314
MOVL C00098 BC00098 V=166.7 PL=0
REFP 3 C00099 BC00099
CALL JOB:SEARCH-R1
SET P0314 P0006
SFTON P0314
MOVL C00100 BC00100 V=166.7 PL=0
SFTOF
'------------------------
MOVL C00101 BC00101 V=333.3
MOVL C00102 BC00102 V=666.7
MOVL C00103 BC00103 V=666.7
MOVL C00104 BC00104 V=666.7
MOVL C00105 BC00105 V=500.0
MOVL C00106 BC00106 V=666.7
MOVL C00107 BC00107 V=666.7
MOVL C00108 BC00108 V=333.3
MOVL C00109 BC00109 V=250.0
'------------------------
'W31.29
'------------------------
MOVL C00110 BC00110 V=166.7 PL=0
REFP 3 C00111 BC00111
CALL JOB:SEARCH-R1
SET P0316 P0006
SFTON P0316
MOVL C00112 BC00112 V=166.7 PL=0
REFP 3 C00113 BC00113
CALL JOB:SEARCH-R1
SET P0316 P0006
SFTON P0316
MOVL C00114 BC00114 V=166.7 PL=0
SFTOF
'------------------------
'W31.31
'------------------------
MOVL C00115 BC00115 V=500.0
MOVL C00116 BC00116 V=166.7 PL=0
REFP 3 C00117 BC00117
CALL JOB:SEARCH-R1
SET P0317 P0006
SFTON P0317
MOVL C00118 BC00118 V=166.7 PL=0
REFP 3 C00119 BC00119
CALL JOB:SEARCH-R1
SET P0317 P0006
SFTON P0317
MOVL C00120 BC00120 V=166.7 PL=0
SFTOF
'------------------------
'W31.32
'------------------------
MOVL C00121 BC00121 V=333.3
MOVL C00122 BC00122 V=333.3
MOVL C00123 BC00123 V=666.7
MOVJ C00124 BC00124 VJ=50.00
MOVJ C00125 BC00125 VJ=50.00
MOVJ C00126 BC00126 VJ=50.00
'W214A P
'------------------------
MOVJ C00127 BC00127 VJ=40.00
MOVL C00128 BC00128 V=166.7 PL=0
REFP 3 C00129 BC00129
CALL JOB:SEARCH-R1
IMOV P0058 V=16.7
SET P0351 P0006
SFTON P0351
REFP 3 C00130 BC00130
CALL JOB:SEARCH-R1
SET P0351 P0006
SFTON P0351
MOVL C00131 BC00131 V=166.7 PL=0
SFTOF
'------------------------
'W219B L
'------------------------
MOVJ C00132 BC00132 VJ=40.00
MOVL C00133 BC00133 V=166.7 PL=0
REFP 3 C00134 BC00134
CALL JOB:SEARCH-R1
IMOV P0058 V=16.7
SET P0352 P0006
SFTON P0352
REFP 3 C00135 BC00135
CALL JOB:SEARCH-R1
SET P0352 P0006
SFTON P0352
MOVL C00136 BC00136 V=166.7 PL=0
SFTOF
'------------------------
'W219B P
'------------------------
MOVJ C00137 BC00137 VJ=40.00
MOVL C00138 BC00138 V=166.7 PL=0
REFP 3 C00139 BC00139
CALL JOB:SEARCH-R1
IMOV P0058 V=16.7
SET P0353 P0006
SFTON P0353
REFP 3 C00140 BC00140
CALL JOB:SEARCH-R1
SET P0353 P0006
SFTON P0353
MOVL C00141 BC00141 V=166.7 PL=0
SFTOF
'------------------------
'W213B L
'------------------------
MOVJ C00142 BC00142 VJ=40.00
MOVL C00143 BC00143 V=166.7 PL=0
REFP 3 C00144 BC00144
CALL JOB:SEARCH-R1
IMOV P0058 V=16.7
SET P0354 P0006
SFTON P0354
REFP 3 C00145 BC00145
CALL JOB:SEARCH-R1
SET P0354 P0006
SFTON P0354
MOVL C00146 BC00146 V=166.7 PL=0
SFTOF
'------------------------
'W213B P
'------------------------
MOVJ C00147 BC00147 VJ=40.00
MOVL C00148 BC00148 V=166.7 PL=0
REFP 3 C00149 BC00149
CALL JOB:SEARCH-R1
IMOV P0058 V=16.7
SET P0355 P0006
SFTON P0355
REFP 3 C00150 BC00150
CALL JOB:SEARCH-R1
SET P0355 P0006
SFTON P0355
MOVL C00151 BC00151 V=166.7 PL=0
SFTOF
'------------------------
'W218B L
'------------------------
MOVJ C00152 BC00152 VJ=40.00
MOVL C00153 BC00153 V=166.7 PL=0
REFP 3 C00154 BC00154
CALL JOB:SEARCH-R1
IMOV P0058 V=16.7
SET P0356 P0006
SFTON P0356
REFP 3 C00155 BC00155
CALL JOB:SEARCH-R1
SET P0356 P0006
SFTON P0356
MOVL C00156 BC00156 V=166.7 PL=0
SFTOF
'------------------------
'W218B P
'------------------------
MOVJ C00157 BC00157 VJ=40.00
MOVL C00158 BC00158 V=166.7 PL=0
REFP 3 C00159 BC00159
CALL JOB:SEARCH-R1
IMOV P0058 V=16.7
SET P0357 P0006
SFTON P0357
REFP 3 C00160 BC00160
CALL JOB:SEARCH-R1
SET P0357 P0006
SFTON P0357
MOVL C00161 BC00161 V=166.7 PL=0
SFTOF
'------------------------
'W215B L
'------------------------
MOVJ C00162 BC00162 VJ=40.00
MOVL C00163 BC00163 V=166.7 PL=0
REFP 3 C00164 BC00164
CALL JOB:SEARCH-R1
IMOV P0058 V=16.7
SET P0358 P0006
SFTON P0358
REFP 3 C00165 BC00165
CALL JOB:SEARCH-R1
SET P0358 P0006
SFTON P0358
MOVL C00166 BC00166 V=166.7 PL=0
SFTOF
'------------------------
'W215B P
'------------------------
MOVL C00167 BC00167 V=666.7
MOVL C00168 BC00168 V=166.7 PL=0
REFP 3 C00169 BC00169
CALL JOB:SEARCH-R1
IMOV P0058 V=16.7
SET P0359 P0006
SFTON P0359
REFP 3 C00170 BC00170
CALL JOB:SEARCH-R1
SET P0359 P0006
SFTON P0359
MOVL C00171 BC00171 V=166.7 PL=0
SFTOF
COMM '------------------------
COMM 'W217B L
COMM '------------------------
COMM MOVL C00172 BC00172 V=666.7
COMM MOVL C00173 BC00173 V=166.7 PL=0
COMM REFP 3 C00174 BC00174
COMM CALL JOB:SEARCH-R1
COMM IMOV P0058 V=16.7
COMM SET P0360 P0006
COMM SFTON P0360
COMM REFP 3 C00175 BC00175
COMM CALL JOB:SEARCH-R1
COMM SET P0360 P0006
COMM SFTON P0360
COMM MOVL C00176 BC00176 V=166.7 PL=0
COMM SFTOF
COMM '------------------------
COMM 'W217B P
COMM '------------------------
COMM MOVL C00177 BC00177 V=666.7
COMM MOVL C00178 BC00178 V=166.7 PL=0
COMM REFP 3 C00179 BC00179
COMM CALL JOB:SEARCH-R1
COMM IMOV P0058 V=16.7
COMM SET P0361 P0006
COMM SFTON P0361
COMM REFP 3 C00180 BC00180
COMM CALL JOB:SEARCH-R1
COMM SET P0361 P0006
COMM SFTON P0361
COMM MOVL C00181 BC00181 V=166.7 PL=0
COMM SFTOF
COMM MOVL C00182 BC00182 V=333.3
MOVL C00183 BC00183 V=666.7
MOVL C00184 BC00184 V=666.7
MOVJ C00185 BC00185 VJ=50.00
MOVJ C00186 BC00186 VJ=50.00
MOVJ C00187 BC00187 VJ=50.00
CALL JOB:FRONT_SEARCH_-90ST-1_4040
MOVJ C00188 BC00188 VJ=50.00
MOVJ C00189 BC00189 VJ=50.00
MOVJ C00190 BC00190 VJ=50.00
MOVL C00191 BC00191 V=666.7
COMM MOVJ C00192 BC00192 VJ=30.00
COMM '------------------------
COMM 'W31.2
COMM '------------------------
COMM SFTON P0300
COMM MOVL C00193 BC00193 V=333.3
COMM MOVL C00194 BC00194 V=166.7 PL=0
COMM MACRO1 MJ#(0) ARGF10
COMM ARCON
COMM MOVL C00195 BC00195 V=10.8
COMM ARCOF
COMM MOVL C00196 BC00196 V=166.7
COMM SFTOF
COMM '------------------------
COMM 'W31.4
COMM '------------------------
COMM SFTON P0301
COMM MOVL C00197 BC00197 V=666.7
COMM MOVL C00198 BC00198 V=166.7 PL=0
COMM ARCON
COMM MOVL C00199 BC00199 V=10.8
COMM ARCOF
COMM MOVL C00200 BC00200 V=166.7
COMM SFTOF
'------------------------
'W31.6
'------------------------
SFTON P0302
MOVL C00201 BC00201 V=666.7
MOVL C00202 BC00202 V=166.7 PL=0
ARCON
MOVL C00203 BC00203 V=10.8
ARCOF
MOVL C00204 BC00204 V=166.7
SFTOF
'------------------------
'W31.8
'------------------------
SFTON P0303
MOVL C00205 BC00205 V=666.7
MOVL C00206 BC00206 V=166.7 PL=0
ARCON
MOVL C00207 BC00207 V=10.8
ARCOF
MOVL C00208 BC00208 V=166.7
SFTOF
'------------------------
'W31.9
'------------------------
SFTON P0304
MOVL C00209 BC00209 V=666.7
MOVL C00210 BC00210 V=166.7 PL=0
ARCON
MOVL C00211 BC00211 V=10.8
ARCOF
MOVL C00212 BC00212 V=166.7
SFTOF
MOVL C00213 BC00213 V=500.0
MOVL C00214 BC00214 V=500.0
MOVJ C00215 BC00215 VJ=50.00
MOVJ C00216 BC00216 VJ=50.00
MOVJ C00217 BC00217 VJ=50.00
MOVJ C00218 BC00218 VJ=50.00
MOVJ C00219 BC00219 VJ=50.00
MOVL C00220 BC00220 V=666.7
'------------------------
'W213A
'------------------------
SFTON P0355
MOVL C00221 BC00221 V=666.7
MOVL C00222 BC00222 V=166.7 PL=0
MACRO1 MJ#(0) ARGF9
ARCON
SFTOF
SFTON P0354
MOVL C00223 BC00223 V=11.2
ARCOF
MOVL C00224 BC00224 V=333.3
SFTOF
MOVJ C00225 BC00225 VJ=50.00
MOVJ C00226 BC00226 VJ=50.00
MOVJ C00227 BC00227 VJ=50.00
MOVJ C00228 BC00228 VJ=50.00
MOVJ C00229 BC00229 VJ=30.00
MOVJ C00230 BC00230 VJ=20.00
MOVJ C00231 BC00231 VJ=20.00
'5.5.1
'------------------------
'W31.11
'------------------------
SFTON P0305
MOVL C00232 BC00232 V=333.3
MOVL C00233 BC00233 V=166.7 PL=0
MACRO1 MJ#(0) ARGF10
ARCON
MOVL C00234 BC00234 V=10.8
ARCOF
MOVL C00235 BC00235 V=166.7
SFTOF
'------------------------
'W31.13
'------------------------
SFTON P0306
MOVL C00236 BC00236 V=500.0
'SPR CZY W DOBRYM MIEJSCU SPOINA
MOVL C00237 BC00237 V=166.7 PL=0
ARCON
MOVL C00238 BC00238 V=10.8
ARCOF
MOVL C00239 BC00239 V=166.7
SFTOF
'------------------------
'W31.14
'------------------------
SFTON P0307
MOVL C00240 BC00240 V=333.3
MOVL C00241 BC00241 V=166.7 PL=0
ARCON
MOVL C00242 BC00242 V=8.3
ARCOF
MOVL C00243 BC00243 V=166.7
SFTOF
MOVL C00244 BC00244 V=333.3
MOVL C00245 BC00245 V=500.0
MOVJ C00246 BC00246 VJ=30.00
MOVJ C00247 BC00247 VJ=30.00
MOVJ C00248 BC00248 VJ=50.00
MOVJ C00249 BC00249 VJ=50.00
'::::::::::::::::::::::::
'::::::::::::::::::::::::
'::::::::::::::::::::::::
'::::::::::::::::::::::::
'::::::::::::::::::::::::
'::::::::::::::::::::::::
'::::::::::::::::::::::::
MOVJ C00250 BC00250 VJ=50.00
MOVJ C00251 BC00251 VJ=50.00
'------------------------
'W214A
'------------------------
SFTON P0351
MOVL C00252 BC00252 V=500.0
MOVL C00253 BC00253 V=166.7 PL=0
MACRO1 MJ#(0) ARGF9
ARCON
MOVL C00254 BC00254 V=11.7
MOVL C00255 BC00255 V=11.0
ARCOF
MOVL C00256 BC00256 V=200.0
SFTOF
MOVJ C00257 BC00257 VJ=50.00
MOVJ C00258 BC00258 VJ=50.00
MOVJ C00259 BC00259 VJ=50.00
MOVJ C00260 BC00260 VJ=40.00
MOVJ C00261 BC00261 VJ=50.00
MOVJ C00262 BC00262 VJ=30.00
MOVJ C00263 BC00263 VJ=30.00
MOVJ C00264 BC00264 VJ=30.00
MOVJ C00265 BC00265 VJ=30.00
'------------------------
'W31.16
'------------------------
SFTON P0308
MOVL C00266 BC00266 V=666.7
MOVL C00267 BC00267 V=166.7 PL=0
MACRO1 MJ#(0) ARGF10
ARCON
MOVL C00268 BC00268 V=10.8
ARCOF
MOVL C00269 BC00269 V=166.7
SFTOF
MOVL C00270 BC00270 V=666.7
MOVL C00271 BC00271 V=666.7
MOVL C00272 BC00272 V=666.7
MOVL C00273 BC00273 V=833.3
MOVL C00274 BC00274 V=666.7
MOVL C00275 BC00275 V=666.7
MOVL C00276 BC00276 V=333.3
MOVL C00277 BC00277 V=333.3
MOVL C00278 BC00278 V=250.0
MOVL C00279 BC00279 V=333.3
'------------------------
'W31.18
'------------------------
SFTON P0309
MOVL C00280 BC00280 V=166.7
MOVL C00281 BC00281 V=83.3 PL=0
ARCON
MOVL C00282 BC00282 V=10.8
ARCOF
MOVL C00283 BC00283 V=166.7
SFTOF
'------------------------
'W31.19
'------------------------
SFTON P0310
MOVL C00284 BC00284 V=333.3
MOVL C00285 BC00285 V=166.7 PL=0
ARCON
MOVL C00286 BC00286 V=10.8
ARCOF
MOVL C00287 BC00287 V=166.7
SFTOF
MOVL C00288 BC00288 V=333.3
MOVL C00289 BC00289 V=500.0
MOVL C00290 BC00290 V=666.7
MOVL C00291 BC00291 V=666.7
MOVJ C00292 BC00292 VJ=40.00
MOVJ C00293 BC00293 VJ=40.00
MOVJ C00294 BC00294 VJ=50.00
'::::::::::::::::::::::::
'::::::::::::::::::::::::
'::::::::::::::::::::::::
'::::::::::::::::::::::::
'::::::::::::::::::::::::
'::::::::::::::::::::::::
'::::::::::::::::::::::::
MOVJ C00295 BC00295 VJ=50.00
MOVJ C00296 BC00296 VJ=50.00
'------------------------
'W215A
'------------------------
SFTON P0359
MOVL C00297 BC00297 V=666.7
MOVL C00298 BC00298 V=166.7 PL=0
MACRO1 MJ#(0) ARGF9
ARCON
SFTOF
SFTON P0358
MOVL C00299 BC00299 V=11.7
ARCOF
MOVL C00300 BC00300 V=333.3
SFTOF
MOVJ C00301 BC00301 VJ=50.00
MOVJ C00302 BC00302 VJ=50.00
MOVJ C00303 BC00303 VJ=50.00
MOVJ C00304 BC00304 VJ=50.00
MOVJ C00305 BC00305 VJ=50.00
MOVJ C00306 BC00306 VJ=50.00
MOVJ C00307 BC00307 VJ=50.00
MOVL C00308 BC00308 V=500.0
'------------------------
'W31.21
'------------------------
SFTON P0311
MOVL C00309 BC00309 V=333.3
MOVL C00310 BC00310 V=166.7 PL=0
MACRO1 MJ#(0) ARGF10
ARCON
MOVL C00311 BC00311 V=10.8
ARCOF
MOVL C00312 BC00312 V=166.7
SFTOF
'------------------------
'W31.22
'------------------------
SFTON P0312
MOVL C00313 BC00313 V=666.7
MOVL C00314 BC00314 V=166.7 PL=0
ARCON
MOVL C00315 BC00315 V=10.8
ARCOF
MOVL C00316 BC00316 V=166.7
SFTOF
'------------------------
'W31.24
'------------------------
SFTON P0313
MOVL C00317 BC00317 V=666.7
MOVL C00318 BC00318 V=166.7 PL=0
ARCON
MOVL C00319 BC00319 V=10.8
ARCOF
SFTOF
MOVL C00320 BC00320 V=166.7
MOVL C00321 BC00321 V=166.7
MOVL C00322 BC00322 V=333.3
SFTOF
MOVL C00323 BC00323 V=333.3
MOVJ C00324 BC00324 VJ=30.00
MOVJ C00325 BC00325 VJ=30.00
MOVJ C00326 BC00326 VJ=50.00
MOVJ C00327 BC00327 VJ=50.00
MOVJ C00328 BC00328 VJ=50.00
COMM '------------------------
COMM 'W215A
COMM '------------------------
COMM MOVJ C00329 BC00329 VJ=50.00
COMM MOVJ C00330 BC00330 VJ=50.00
COMM SFTON P0360
COMM MOVL C00331 BC00331 V=500.0
COMM MOVL C00332 BC00332 V=500.0
COMM MOVL C00333 BC00333 V=166.7 PL=0
COMM MACRO1 MJ#(0) ARGF9
COMM ARCON
COMM SFTOF
COMM SFTON P0361
COMM MOVL C00334 BC00334 V=11.7
COMM MOVL C00335 BC00335 V=11.7
COMM ARCOF
COMM MOVL C00336 BC00336 V=500.0
COMM SFTOF
COMM MOVJ C00337 BC00337 VJ=50.00
COMM MOVJ C00338 BC00338 VJ=50.00
COMM MOVJ C00339 BC00339 VJ=50.00
COMM MOVJ C00340 BC00340 VJ=80.00
COMM MOVJ C00341 BC00341 VJ=50.00
MOVJ C00342 BC00342 VJ=50.00
MOVJ C00343 BC00343 VJ=40.00
MOVJ C00344 BC00344 VJ=20.00
MOVL C00345 BC00345 V=333.3
'------------------------
'W31.26
'------------------------
SFTON P0314
MOVL C00346 BC00346 V=833.3
MOVL C00347 BC00347 V=166.7 PL=0
MACRO1 MJ#(0) ARGF10
ARCON
MOVL C00348 BC00348 V=10.8
ARCOF
MOVL C00349 BC00349 V=166.7
SFTOF
'------------------------
MOVL C00350 BC00350 V=500.0
MOVL C00351 BC00351 V=500.0
MOVL C00352 BC00352 V=500.0
MOVL C00353 BC00353 V=500.0
'W31.27
'------------------------
MOVL C00354 BC00354 V=500.0
SFTON P0316
MOVL C00355 BC00355 V=166.7 PL=0
ARCON
MOVL C00356 BC00356 V=10.8
ARCOF
SFTOF
MOVL C00357 BC00357 V=200.0
SFTOF
MOVL C00358 BC00358 V=333.3
MOVL C00359 BC00359 V=416.7
MOVJ C00360 BC00360 VJ=30.00
MOVJ C00361 BC00361 VJ=50.00
MOVJ C00362 BC00362 VJ=50.00
MOVJ C00363 BC00363 VJ=50.00
'------------------------
'W218A
'------------------------
MOVJ C00364 BC00364 VJ=50.00
MOVJ C00365 BC00365 VJ=50.00
SFTON P0357
MOVL C00366 BC00366 V=500.0
MOVL C00367 BC00367 V=500.0
MOVL C00368 BC00368 V=166.7 PL=0
MACRO1 MJ#(0) ARGF9
ARCON
SFTOF
SFTON P0356
MOVL C00369 BC00369 V=11.7
ARCOF
MOVL C00370 BC00370 V=333.3
SFTOF
MOVJ C00371 BC00371 VJ=50.00
MOVJ C00372 BC00372 VJ=50.00
MOVJ C00373 BC00373 VJ=50.00
MOVJ C00374 BC00374 VJ=50.00
MOVJ C00375 BC00375 VJ=50.00
MOVJ C00376 BC00376 VJ=50.00
MOVL C00377 BC00377 V=500.0
'------------------------
'W31.29
'------------------------
SFTON P0317
MOVL C00378 BC00378 V=333.3
MOVL C00379 BC00379 V=333.3
MOVL C00380 BC00380 V=166.7 PL=0
MOVL C00381 BC00381 V=166.7 PL=0
MACRO1 MJ#(0) ARGF10
ARCON
MOVL C00382 BC00382 V=10.8
ARCOF
MOVL C00383 BC00383 V=166.7
SFTOF
'------------------------
'W31.31
'------------------------
'------------------------
'W31.32
'------------------------
SFTON P0317
MOVL C00384 BC00384 V=166.7 PL=0
ARCON
MOVL C00385 BC00385 V=11.0
ARCOF
SFTOF
MOVL C00386 BC00386 V=333.3
MOVL C00387 BC00387 V=416.7
MOVL C00388 BC00388 V=500.0
MOVL C00389 BC00389 V=500.0
MOVL C00390 BC00390 V=500.0
MOVJ C00391 BC00391 VJ=40.00
MOVJ C00392 BC00392 VJ=50.00
MOVJ C00393 BC00393 VJ=50.00
MOVJ C00394 BC00394 VJ=50.00
MOVJ C00395 BC00395 VJ=50.00
MOVJ C00396 BC00396 VJ=50.00
SFTON P0353
MOVL C00397 BC00397 V=666.7
MOVL C00398 BC00398 V=250.0
MOVL C00399 BC00399 V=166.7 PL=0
MACRO1 MJ#(0) ARGF9
ARCON
SFTOF
SFTON P0352
MOVL C00400 BC00400 V=11.7
ARCOF
MOVL C00401 BC00401 V=250.0
SFTOF
MOVJ C00402 BC00402 VJ=50.00
MOVJ C00403 BC00403 VJ=50.00
CALL JOB:FRONT_WELD_-90ST-1_4040
CALL JOB:MOVE_OUT_OF_TUNNEL
END
